(* PLC project flexManufacturing.project, CODESYS CODESYS V3.5 SP16 Patch 3 *)
(* stored: creationDateTime 2021-01-27T23:10:48.5476869, modificationDateTime 2021-01-27T23:10:24.2476033 *)

PROGRAM PLC_PRG
  VAR
    FM_CPS_PP_DETECTED : BOOL;  (* INPUTS *)
    FM_CPS_PP_MOVINGX : BOOL;
    FM_CPS_PP_MOVINGZ : BOOL;
    FM_CPS_PP_ROTATING : BOOL;
    FM_CPS_TRANSFER_END : BOOL;
    FM_INPUT_1_SENSOR : BOOL;
    FM_INPUT_2_SENSOR : BOOL;
    FM_PALLET_1_CONV_1_END : BOOL;
    FM_PALLET_1_CONV_2_END : BOOL;
    FM_PALLET_2_CONV_1_END : BOOL;
    FM_PALLET_2_CONV_6_END : BOOL;
    FM_PALLET_3_CONV_1_END : BOOL;
    FM_PALLET_3_CONV_2_END : BOOL;
    FM_PALLET_4_CONV_1_END : BOOL;
    FM_PALLET_4_CONV_4_END : BOOL;
    FM_PALLET_5_CONV_1_END : BOOL;
    FM_PALLET_5_CONV_3_END : BOOL;
    FM_PALLET_2_CONV_2_3_SENSOR : BOOL;
    FM_PALLET_2_CONV_4_5_SENSOR : BOOL;
    FM_PALLET_4_CONV_2_3_SENSOR : BOOL;
    FM_PALLET_5_CONV_2_3_SENSOR : BOOL;
    FM_WS_1_M_BUSY : BOOL;
    FM_WS_2_M_BUSY : BOOL;
    FM_WS_1_PP_1_MOVINGX : BOOL;
    FM_WS_1_PP_1_MOVINGZ : BOOL;
    FM_WS_1_PP_2_MOVINGX : BOOL;
    FM_WS_1_PP_2_MOVINGZ : BOOL;
    FM_WS_2_PP_1_MOVINGX : BOOL;
    FM_WS_2_PP_1_MOVINGZ : BOOL;
    FM_WS_2_PP_2_MOVINGX : BOOL;
    FM_WS_2_PP_2_MOVINGZ : BOOL;
    FM_WS_3_PP_1_MOVINGX : BOOL;
    FM_WS_3_PP_1_MOVINGZ : BOOL;
    FM_WS_3_PP_2_MOVINGX : BOOL;
    FM_WS_3_PP_2_MOVINGZ : BOOL;
    FM_WS_3_PP_3_MOVINGX : BOOL;
    FM_WS_3_PP_3_MOVINGZ : BOOL;
    FM_WS_3_PP_4_MOVINGX : BOOL;
    FM_WS_3_PP_4_MOVINGZ : BOOL;
    FM_WS_1_PP_1_DETECTED : BOOL;
    FM_WS_1_PP_1_ROTATING : BOOL;
    FM_WS_1_PP_2_DETECTED : BOOL;
    FM_WS_1_PP_2_ROTATING : BOOL;
    FM_WS_2_PP_1_DETECTED : BOOL;
    FM_WS_2_PP_1_ROTATING : BOOL;
    FM_WS_2_PP_2_DETECTED : BOOL;
    FM_WS_2_PP_2_ROTATING : BOOL;
    FM_WS_3_PP_1_DETECTED : BOOL;
    FM_WS_3_PP_1_ROTATING : BOOL;
    FM_WS_3_PP_2_DETECTED : BOOL;
    FM_WS_3_PP_2_ROTATING : BOOL;
    FM_WS_3_PP_3_DETECTED : BOOL;
    FM_WS_3_PP_3_ROTATING : BOOL;
    FM_WS_3_PP_4_DETECTED : BOOL;
    FM_WS_3_PP_4_ROTATING : BOOL;
    FM_ZONE_1_SENSOR_1 : BOOL;
    FM_ZONE_1_SENSOR_2 : BOOL;
    FM_ZONE_2_SENSOR_1 : BOOL;
    FM_ZONE_2_SENSOR_2 : BOOL;
    FM_ZONE_3_SENSOR_1 : BOOL;
    FM_ZONE_3_SENSOR_2 : BOOL;
    FM_ZONE_4_SENSOR_1 : BOOL;
    FM_ZONE_4_SENSOR_2 : BOOL;
    FM_WS_3_CONV_PROD_END : BOOL;
    FM_CPS_CONV_F : BOOL;  (* OUTPUTS *)
    FM_CPS_INBOX_F : BOOL;
    FM_CPS_INBOX_WARNINGL : BOOL;
    FM_CPS_OUT_WARNINGl : BOOL;
    FM_CPS_PP_GRAB : BOOL;
    FM_CPS_PP_MOVX : BOOL;
    FM_CPS_PP_MOVZ : BOOL;
    FM_CPS_PP_ROTCW : BOOL;
    FM_CPS_PP_ROTCCW : BOOL;
    FM_CPS_TRANSFER_F : BOOL;
    FM_CPS_TRANSFER_R : BOOL;
    FM_INPUT_1 : BOOL;
    FM_INPUT_2 : BOOL;
    FM_INPUT_1_WARNINGL : BOOL;
    FM_INPUT_2_WARNINGL : BOOL;
    FM_PALLET_1_CONV_1_B : BOOL;
    FM_PALLET_1_CONV_1_F : BOOL;
    FM_PALLET_1_CONV_2_B : BOOL;
    FM_PALLET_1_CONV_2_F : BOOL;
    FM_PALLET_2_CONV_1_B : BOOL;
    FM_PALLET_2_CONV_1_F : BOOL;
    FM_PALLET_2_CONV_2_B : BOOL;
    FM_PALLET_2_CONV_2_F : BOOL;
    FM_PALLET_2_CONV_3_B : BOOL;
    FM_PALLET_2_CONV_3_F : BOOL;
    FM_PALLET_2_CONV_6_B : BOOL;
    FM_PALLET_2_CONV_6_F : BOOL;
    FM_PALLET_3_CONV_1_B : BOOL;
    FM_PALLET_3_CONV_1_F : BOOL;
    FM_PALLET_3_CONV_2_B : BOOL;
    FM_PALLET_3_CONV_2_F : BOOL;
    FM_PALLET_4_CONV_1_B : BOOL;
    FM_PALLET_4_CONV_1_F : BOOL;
    FM_PALLET_5_CONV_3_B : BOOL;
    FM_PALLET_5_CONV_3_F : BOOL;
    FM_PALLET_2_CONV_4_B_0 : BOOL;
    FM_PALLET_2_CONV_4_B_1 : BOOL;
    FM_PALLET_2_CONV_4_B_2 : BOOL;
    FM_PALLET_2_CONV_4_F_0 : BOOL;
    FM_PALLET_2_CONV_4_F_1 : BOOL;
    FM_PALLET_2_CONV_4_F_2 : BOOL;
    FM_PALLET_2_CONV_5_B_0 : BOOL;
    FM_PALLET_2_CONV_5_B_1 : BOOL;
    FM_PALLET_2_CONV_5_B_2 : BOOL;
    FM_PALLET_2_CONV_5_F_0 : BOOL;
    FM_PALLET_2_CONV_5_F_1 : BOOL;
    FM_PALLET_2_CONV_5_F_2 : BOOL;
    FM_PALLET_4_CONV_2_B_0 : BOOL;
    FM_PALLET_4_CONV_2_B_1 : BOOL;
    FM_PALLET_4_CONV_2_B_2 : BOOL;
    FM_PALLET_4_CONV_2_F_0 : BOOL;
    FM_PALLET_4_CONV_2_F_1 : BOOL;
    FM_PALLET_4_CONV_2_F_2 : BOOL;
    FM_PALLET_4_CONV_3_B_0 : BOOL;
    FM_PALLET_4_CONV_3_B_1 : BOOL;
    FM_PALLET_4_CONV_3_B_2 : BOOL;
    FM_PALLET_4_CONV_3_F_0 : BOOL;
    FM_PALLET_4_CONV_3_F_1 : BOOL;
    FM_PALLET_4_CONV_3_F_2 : BOOL;
    FM_PALLET_4_CONV_4_B_0 : BOOL;
    FM_PALLET_4_CONV_4_B_1 : BOOL;
    FM_PALLET_4_CONV_4_B_2 : BOOL;
    FM_PALLET_4_CONV_4_F_0 : BOOL;
    FM_PALLET_4_CONV_4_F_1 : BOOL;
    FM_PALLET_4_CONV_4_F_2 : BOOL;
    FM_PALLET_5_CONV_1_B_0 : BOOL;
    FM_PALLET_5_CONV_1_B_1 : BOOL;
    FM_PALLET_5_CONV_1_B_2 : BOOL;
    FM_PALLET_5_CONV_1_F_0 : BOOL;
    FM_PALLET_5_CONV_1_F_1 : BOOL;
    FM_PALLET_5_CONV_1_F_2 : BOOL;
    FM_PALLET_5_CONV_2_B_0 : BOOL;
    FM_PALLET_5_CONV_2_B_1 : BOOL;
    FM_PALLET_5_CONV_2_F_0 : BOOL;
    FM_PALLET_5_CONV_2_F_1 : BOOL;
    FM_WS_1_M_START : BOOL;
    FM_WS_2_M_START : BOOL;
    FM_WS_1_WARNINGL : BOOL;
    FM_WS_2_WARNINGL : BOOL;
    FM_WS_1_PP_1_GRAB : BOOL;
    FM_WS_1_PP_1_MOVX : BOOL;
    FM_WS_1_PP_1_MOVZ : BOOL;
    FM_WS_1_PP_2_GRAB : BOOL;
    FM_WS_1_PP_2_MOVX : BOOL;
    FM_WS_1_PP_2_MOVZ : BOOL;
    FM_WS_2_PP_1_GRAB : BOOL;
    FM_WS_2_PP_1_MOVX : BOOL;
    FM_WS_2_PP_1_MOVZ : BOOL;
    FM_WS_2_PP_2_GRAB : BOOL;
    FM_WS_2_PP_2_MOVX : BOOL;
    FM_WS_2_PP_2_MOVZ : BOOL;
    FM_WS_3_CONV_PROD : BOOL;
    FM_WS_3_PP_1_GRAB : BOOL;
    FM_WS_3_PP_1_MOVX : BOOL;
    FM_WS_3_PP_1_MOVZ : BOOL;
    FM_WS_3_PP_2_GRAB : BOOL;
    FM_WS_3_PP_2_MOVX : BOOL;
    FM_WS_3_PP_2_MOVZ : BOOL;
    FM_WS_3_PP_3_GRAB : BOOL;
    FM_WS_3_PP_3_MOVX : BOOL;
    FM_WS_3_PP_3_MOVZ : BOOL;
    FM_WS_3_PP_4_GRAB : BOOL;
    FM_WS_3_PP_4_MOVX : BOOL;
    FM_WS_3_PP_4_MOVZ : BOOL;
    FM_WS_1_PP_1_ROTCW : BOOL;
    FM_WS_1_PP_2_ROTCW : BOOL;
    FM_WS_2_PP_1_ROTCW : BOOL;
    FM_WS_2_PP_2_ROTCW : BOOL;
    FM_WS_3_CONV_LID_0 : BOOL;
    FM_WS_3_CONV_LID_1 : BOOL;
    FM_WS_3_CONV_LID_2 : BOOL;
    FM_WS_3_CONV_LID_END : BOOL;
    FM_WS_3_PP_1_ROTCW : BOOL;
    FM_WS_3_PP_2_ROTCW : BOOL;
    FM_WS_3_PP_3_ROTCW : BOOL;
    FM_WS_3_PP_4_ROTCW : BOOL;
    FM_WS_1_PP_1_ROTCCW : BOOL;
    FM_WS_1_PP_2_ROTCCW : BOOL;
    FM_WS_2_PP_1_ROTCCW : BOOL;
    FM_WS_2_PP_2_ROTCCW : BOOL;
    FM_WS_3_CONV_BASE_0 : BOOL;
    FM_WS_3_CONV_BASE_1 : BOOL;
    FM_WS_3_CONV_BASE_2 : BOOL;
    FM_WS_3_CONV_BASE_3 : BOOL;
    FM_WS_3_CONV_BASE_END : BOOL;
    FM_WS_3_PP_1_ROTCCW : BOOL;
    FM_WS_3_PP_2_ROTCCW : BOOL;
    FM_WS_3_PP_3_ROTCCW : BOOL;
    FM_WS_3_PP_4_ROTCCW : BOOL;
    WS_1_PP_1_FALLEDGE : F_TRIG;
    WS_1_PP_1_STEP : INT := 0;
    WS_1_PP_1_TON : TON;
    WS_1_PP_2_FALLEDGE : F_TRIG;
    WS_1_PP_2_STEP : INT := 0;
    WS_1_PP_2_TON : TON;
    WS_2_PP_1_FALLEDGE : F_TRIG;
    WS_2_PP_1_STEP : INT := 0;
    WS_2_PP_1_TON : TON;
    WS_2_PP_2_FALLEDGE : F_TRIG;
    WS_2_PP_2_STEP : INT := 0;
    WS_2_PP_2_TON : TON;
    WS_3_PP_1_FALLEDGE : F_TRIG;
    WS_3_PP_1_STEP : INT := 0;
    WS_3_PP_1_TON : TON;
    WS_3_PP_2_FALLEDGE : F_TRIG;
    WS_3_PP_2_STEP : INT := 0;
    WS_3_PP_2_TON : TON;
    WS_3_PP_3_FALLEDGE : F_TRIG;
    WS_3_PP_3_STEP : INT := 0;
    WS_3_PP_3_TON : TON;
    WS_3_PP_4_FALLEDGE : F_TRIG;
    WS_3_PP_4_STEP : INT := 0;
    WS_3_PP_4_TON : TON;
    WS_3_RESET_FALLEDGE : F_TRIG;
    WS_3_RESET_STEP : INT := 0;
    WS_3_RESET_TON : TON;
    CPS_PP_FALLEDGE : F_TRIG;
    CPS_PP_STEP : INT := 0;
    CPS_PP_TON : TON;
    CPS_RESET_FALLEDGE : F_TRIG;
    CPS_RESET_STEP : INT := 0;
    CPS_RESET_TON : TON;
    P_1_CONV_1_END_F : F_TRIG;
    P_1_CONV_2_END_F : F_TRIG;
    P_2_CONV_1_END_F : F_TRIG;
    P_2_CONV_6_END_F : F_TRIG;
    P_3_CONV_1_END_F : F_TRIG;
    TR_T3 : BOOL;
    TR_T2 : BOOL;
    TR_T7 : BOOL;
    TR_T10 : BOOL;
    TR_T11 : BOOL;
    TR_T6 : BOOL;
    TR_T15 : BOOL;
    TR_T14 : BOOL;
    TR_T19 : BOOL;
    TR_T18 : BOOL;
  END_VAR

(* transition INPUT_1_TR_FALL *)
                        P_1_CONV_1_END_F(CLK:=FM_PALLET_1_CONV_1_END);
INPUT_1_TR_FALL:=P_1_CONV_1_END_F.Q;
                      
(* transition P_1_C_2_END_TR_F *)
                        P_1_CONV_2_END_F(CLK:=FM_PALLET_1_CONV_2_END);
P_1_C_2_END_TR_F:=P_1_CONV_2_END_F.Q;
                      
(* transition P_2_C_6_END_TR_F *)
                        P_2_CONV_6_END_F(CLK:=FM_PALLET_2_CONV_6_END);
P_2_C_6_END_TR_F:=P_2_CONV_6_END_F.Q;
                      
(* transition INPUT_2_TR_FALL *)
                        P_2_CONV_1_END_F(CLK:=FM_PALLET_2_CONV_1_END);
INPUT_2_TR_FALL:=P_2_CONV_1_END_F.Q;
                      
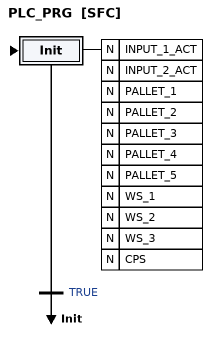
INITIAL_STEP Init:
  INPUT_1_ACT(N);
  INPUT_2_ACT(N);
  PALLET_1(N);
  PALLET_2(N);
  PALLET_3(N);
  PALLET_4(N);
  PALLET_5(N);
  WS_1(N);
  WS_2(N);
  WS_3(N);
  CPS(N);
END_STEP
TRANSITION FROM Init TO Init
  := TRUE;
END_TRANSITION

ACTION WS_1_ACT_PP_1:
                        
CASE WS_1_PP_1_STEP OF
	
	0:	FM_WS_1_PP_1_MOVX:=TRUE;
		WS_1_PP_1_STEP:=1;
		
	1:	FM_WS_1_PP_1_ROTCW:=TRUE;
		WS_1_PP_1_STEP:=2;
	
	2:	WS_1_PP_1_FALLEDGE(CLK:=FM_WS_1_PP_1_ROTATING);
		WHILE WS_1_PP_1_FALLEDGE.Q DO
			FM_WS_1_PP_1_MOVZ:=TRUE;
			WS_1_PP_1_STEP:=3;
			WS_1_PP_1_FALLEDGE(CLK:=FALSE);
		END_WHILE
		
	3:	FM_WS_1_PP_1_GRAB:=TRUE;
		WS_1_PP_1_STEP:=4;
		
	4:	WS_1_PP_1_FALLEDGE(CLK:=FM_WS_1_PP_1_MOVINGZ);
		WHILE WS_1_PP_1_FALLEDGE.Q DO
			FM_WS_1_PP_1_MOVZ:=FALSE;
			WS_1_PP_1_STEP:=5;
			WS_1_PP_1_FALLEDGE(CLK:=FALSE);
		END_WHILE
		
	5:	WS_1_PP_1_FALLEDGE(CLK:=FM_WS_1_PP_1_MOVINGZ);
		WHILE WS_1_PP_1_FALLEDGE.Q DO
			FM_WS_1_PP_1_ROTCCW:=TRUE;
			WS_1_PP_1_STEP:=6;
			WS_1_PP_1_FALLEDGE(CLK:=FALSE);
		END_WHILE
		
	6:	WS_1_PP_1_FALLEDGE(CLK:=FM_WS_1_PP_1_ROTATING);
		WHILE WS_1_PP_1_FALLEDGE.Q DO
			WS_1_PP_1_STEP:=7;
			WS_1_PP_1_FALLEDGE(CLK:=FALSE);
		END_WHILE
		
	7:	WS_1_PP_1_TON(IN:=TRUE,PT:=T#1S);
		WHILE WS_1_PP_1_TON.Q DO
			FM_WS_1_PP_1_GRAB:=FALSE;
			WS_1_PP_1_STEP:=8;
			WS_1_PP_1_TON(IN:=FALSE);
		END_WHILE
		
	8:	WS_1_PP_1_TON(IN:=TRUE,PT:=T#1S);
		WHILE WS_1_PP_1_TON.Q DO
			WS_1_PP_1_STEP:=9;
			WS_1_PP_1_TON(IN:=FALSE);
		END_WHILE
		
	9:	WS_1_PP_1_STEP:=0;
	
END_CASE

                      
END_ACTION

ACTION WS_1:
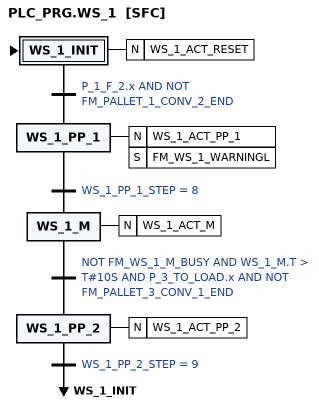
INITIAL_STEP WS_1_INIT:
  WS_1_ACT_RESET(N);
END_STEP
TRANSITION FROM WS_1_INIT TO WS_1_PP_1
  := P_1_F_2.x AND NOT FM_PALLET_1_CONV_2_END;
END_TRANSITION
STEP WS_1_PP_1:
  WS_1_ACT_PP_1(N);
  FM_WS_1_WARNINGL(S);
END_STEP
TRANSITION FROM WS_1_PP_1 TO WS_1_M
  := WS_1_PP_1_STEP = 8;
END_TRANSITION
STEP WS_1_M:
  WS_1_ACT_M(N);
END_STEP
TRANSITION FROM WS_1_M TO WS_1_PP_2
  := NOT FM_WS_1_M_BUSY AND WS_1_M.T > T#10S AND P_3_TO_LOAD.x AND NOT FM_PALLET_3_CONV_1_END;
END_TRANSITION
STEP WS_1_PP_2:
  WS_1_ACT_PP_2(N);
END_STEP
TRANSITION FROM WS_1_PP_2 TO WS_1_INIT
  := WS_1_PP_2_STEP = 9;
END_TRANSITION
END_ACTION

ACTION WS_1_ACT_PP_2:
                        
CASE WS_1_PP_2_STEP OF
	
	0:	FM_WS_1_PP_2_MOVX:=TRUE;
		WS_1_PP_2_STEP:=1;
		
	1:	WS_1_PP_2_FALLEDGE(CLK:=FM_WS_1_PP_2_MOVINGX);
		WHILE WS_1_PP_2_FALLEDGE.Q DO
			FM_WS_1_PP_2_MOVZ:=TRUE;
			WS_1_PP_2_STEP:=2;
			WS_1_PP_2_FALLEDGE(CLK:=FALSE);
		END_WHILE
		
	2:	FM_WS_1_PP_2_GRAB:=TRUE;
		WS_1_PP_2_STEP:=3;
		
	3:	WS_1_PP_2_FALLEDGE(CLK:=FM_WS_1_PP_2_MOVINGZ);
		WHILE WS_1_PP_2_FALLEDGE.Q DO
			FM_WS_1_PP_2_MOVZ:=FALSE;
			WS_1_PP_2_STEP:=4;
			WS_1_PP_2_FALLEDGE(CLK:=FALSE);
		END_WHILE
		
	4:	WS_1_PP_2_FALLEDGE(CLK:=FM_WS_1_PP_2_MOVINGZ);
		WHILE WS_1_PP_2_FALLEDGE.Q DO
			FM_WS_1_PP_2_ROTCCW:=TRUE;
			WS_1_PP_2_STEP:=5;
			WS_1_PP_2_FALLEDGE(CLK:=FALSE);
		END_WHILE
		
	5:	WS_1_PP_2_FALLEDGE(CLK:=FM_WS_1_PP_2_ROTATING);
		WHILE WS_1_PP_2_FALLEDGE.Q DO
			WS_1_PP_2_STEP:=6;
			FM_WS_1_PP_2_ROTCCW:=FALSE;
			WS_1_PP_2_FALLEDGE(CLK:=FALSE);
		END_WHILE
		
	6:	WS_1_PP_2_TON(IN:=TRUE,PT:=T#1S);
		WHILE WS_1_PP_2_TON.Q DO
			FM_WS_1_PP_2_GRAB:=FALSE;
			WS_1_PP_2_STEP:=7;
			WS_1_PP_2_TON(IN:=FALSE);
		END_WHILE
		
	7:	WS_1_PP_2_TON(IN:=TRUE,PT:=T#1S);
		WHILE WS_1_PP_2_TON.Q DO
			FM_WS_1_PP_2_ROTCW:=TRUE;
			WS_1_PP_2_STEP:=8;
			WS_1_PP_2_TON(IN:=FALSE);
		END_WHILE
		
	8:	WS_1_PP_2_FALLEDGE(CLK:=FM_WS_1_PP_2_ROTATING);
		WHILE WS_1_PP_2_FALLEDGE.Q DO
			WS_1_PP_2_STEP:=9;
			FM_WS_1_PP_2_ROTCW:=FALSE;
			WS_1_PP_2_FALLEDGE(CLK:=FALSE);
		END_WHILE
		
	9: WS_1_PP_2_STEP:=0;
END_CASE
                      
END_ACTION

ACTION WS_1_ACT_M:
                        FM_WS_1_M_START:=TRUE;
                      
END_ACTION

ACTION WS_1_ACT_RESET:
                        FM_WS_1_PP_1_MOVX:=FALSE;
FM_WS_1_PP_1_ROTCCW:=FALSE;
FM_WS_1_PP_1_ROTCW:=FALSE;
FM_WS_1_M_START:=FALSE;
FM_WS_1_WARNINGL:=FALSE;
FM_WS_1_PP_2_MOVX:=FALSE;
FM_WS_1_PP_2_ROTCCW:=FALSE;
FM_WS_1_PP_2_ROTCW:=FALSE;

                      
END_ACTION

ACTION WS_3:
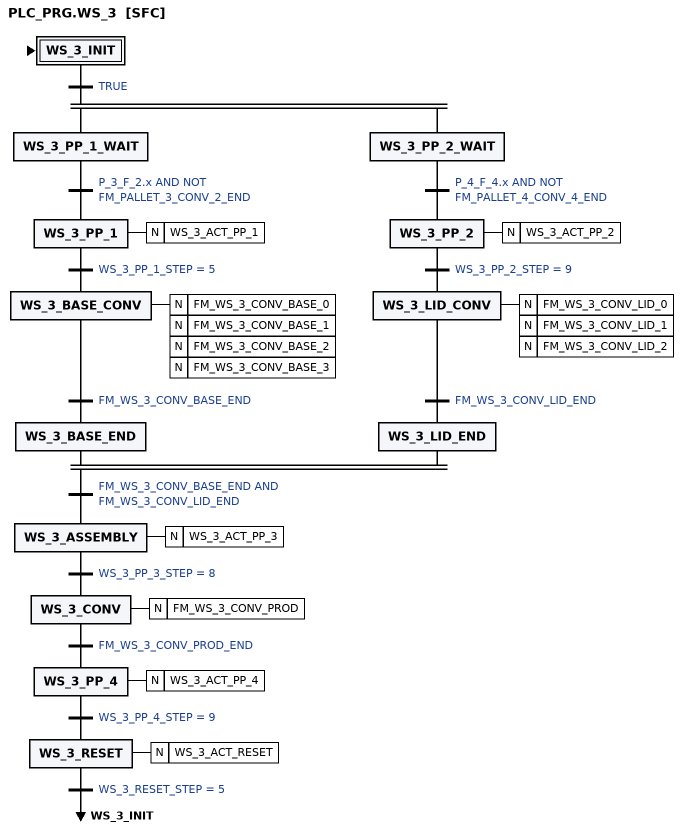
INITIAL_STEP WS_3_INIT:
END_STEP
TRANSITION FROM WS_3_INIT TO (WS_3_PP_1_WAIT, WS_3_PP_2_WAIT)
  := TRUE;
END_TRANSITION
STEP WS_3_PP_1_WAIT:
END_STEP
TRANSITION FROM WS_3_PP_1_WAIT TO WS_3_PP_1
  := P_3_F_2.x AND NOT FM_PALLET_3_CONV_2_END;
END_TRANSITION
STEP WS_3_PP_1:
  WS_3_ACT_PP_1(N);
END_STEP
TRANSITION FROM WS_3_PP_1 TO WS_3_BASE_CONV
  := WS_3_PP_1_STEP = 5;
END_TRANSITION
STEP WS_3_BASE_CONV:
  FM_WS_3_CONV_BASE_0(N);
  FM_WS_3_CONV_BASE_1(N);
  FM_WS_3_CONV_BASE_2(N);
  FM_WS_3_CONV_BASE_3(N);
END_STEP
TRANSITION FROM WS_3_BASE_CONV TO WS_3_BASE_END
  := FM_WS_3_CONV_BASE_END;
END_TRANSITION
STEP WS_3_BASE_END:
END_STEP
TRANSITION FROM (WS_3_BASE_END, WS_3_LID_END) TO WS_3_ASSEMBLY
  := FM_WS_3_CONV_BASE_END AND FM_WS_3_CONV_LID_END;
END_TRANSITION
STEP WS_3_PP_2_WAIT:
END_STEP
TRANSITION FROM WS_3_PP_2_WAIT TO WS_3_PP_2
  := P_4_F_4.x AND NOT FM_PALLET_4_CONV_4_END;
END_TRANSITION
STEP WS_3_PP_2:
  WS_3_ACT_PP_2(N);
END_STEP
TRANSITION FROM WS_3_PP_2 TO WS_3_LID_CONV
  := WS_3_PP_2_STEP = 9;
END_TRANSITION
STEP WS_3_LID_CONV:
  FM_WS_3_CONV_LID_0(N);
  FM_WS_3_CONV_LID_1(N);
  FM_WS_3_CONV_LID_2(N);
END_STEP
TRANSITION FROM WS_3_LID_CONV TO WS_3_LID_END
  := FM_WS_3_CONV_LID_END;
END_TRANSITION
STEP WS_3_LID_END:
END_STEP
STEP WS_3_ASSEMBLY:
  WS_3_ACT_PP_3(N);
END_STEP
TRANSITION FROM WS_3_ASSEMBLY TO WS_3_CONV
  := WS_3_PP_3_STEP = 8;
END_TRANSITION
STEP WS_3_CONV:
  FM_WS_3_CONV_PROD(N);
END_STEP
TRANSITION FROM WS_3_CONV TO WS_3_PP_4
  := FM_WS_3_CONV_PROD_END;
END_TRANSITION
STEP WS_3_PP_4:
  WS_3_ACT_PP_4(N);
END_STEP
TRANSITION FROM WS_3_PP_4 TO WS_3_RESET
  := WS_3_PP_4_STEP = 9;
END_TRANSITION
STEP WS_3_RESET:
  WS_3_ACT_RESET(N);
END_STEP
TRANSITION FROM WS_3_RESET TO WS_3_INIT
  := WS_3_RESET_STEP = 5;
END_TRANSITION
END_ACTION

ACTION WS_3_ACT_PP_1:
                        
CASE WS_3_PP_1_STEP OF
	
	0:	FM_WS_3_PP_1_MOVZ:=TRUE;
		FM_WS_3_PP_1_GRAB:=TRUE;
		WS_3_PP_1_STEP:=1;
		
	1:	WS_3_PP_1_FALLEDGE(CLK:=FM_WS_3_PP_1_MOVINGZ);
		WHILE WS_3_PP_1_FALLEDGE.Q DO
			FM_WS_3_PP_1_MOVZ:=FALSE;
			WS_3_PP_1_STEP:=2;
			WS_3_PP_1_FALLEDGE(CLK:=FALSE);
		END_WHILE
	
	2:	WS_3_PP_1_FALLEDGE(CLK:=FM_WS_3_PP_1_MOVINGZ);
		WHILE WS_3_PP_1_FALLEDGE.Q DO
			FM_WS_3_PP_1_MOVX:=TRUE;
			WS_3_PP_1_STEP:=3;
			WS_3_PP_1_FALLEDGE(CLK:=FALSE);
		END_WHILE
		
	3:	WS_3_PP_1_FALLEDGE(CLK:=FM_WS_3_PP_1_MOVINGX);
		WHILE WS_3_PP_1_FALLEDGE.Q DO
			WS_3_PP_1_STEP:=4;
			WS_3_PP_1_FALLEDGE(CLK:=FALSE);
		END_WHILE
		
	4:	WS_3_PP_1_TON(IN:=TRUE,PT:=T#200MS);
		WHILE WS_3_PP_1_TON.Q DO
			FM_WS_3_PP_1_GRAB:=FALSE;
			WS_3_PP_1_STEP:=5;
			WS_3_PP_1_TON(IN:=FALSE);
		END_WHILE
		
	5:	WS_3_PP_1_STEP:=0;
	
END_CASE
                      
END_ACTION

ACTION WS_3_ACT_PP_2:
                        
CASE WS_3_PP_2_STEP OF
	
	0:	FM_WS_3_PP_2_MOVX:=TRUE;
		WS_3_PP_2_STEP:=1;
		
	1:	WS_3_PP_2_FALLEDGE(CLK:=FM_WS_3_PP_2_MOVINGX);
		WHILE WS_3_PP_2_FALLEDGE.Q DO
			FM_WS_3_PP_2_MOVZ:=TRUE;
			FM_WS_3_PP_2_GRAB:=TRUE;
			WS_3_PP_2_STEP:=2;
			WS_3_PP_2_FALLEDGE(CLK:=FALSE);
		END_WHILE
	
	2:	WS_3_PP_2_FALLEDGE(CLK:=FM_WS_3_PP_2_MOVINGZ);
		WHILE WS_3_PP_2_FALLEDGE.Q DO
			FM_WS_3_PP_2_MOVZ:=FALSE;
			WS_3_PP_2_STEP:=3;
			WS_3_PP_2_FALLEDGE(CLK:=FALSE);
		END_WHILE
		
	3:	WS_3_PP_2_FALLEDGE(CLK:=FM_WS_3_PP_2_MOVINGZ);
		WHILE WS_3_PP_2_FALLEDGE.Q DO
			FM_WS_3_PP_2_ROTCCW:=TRUE;
			WS_3_PP_2_STEP:=4;
			WS_3_PP_2_FALLEDGE(CLK:=FALSE);
		END_WHILE
		
	4:	WS_3_PP_2_FALLEDGE(CLK:=FM_WS_3_PP_2_ROTATING);
		WHILE WS_3_PP_2_FALLEDGE.Q DO
			FM_WS_3_PP_2_ROTCCW:=FALSE;
			WS_3_PP_2_STEP:=5;
			WS_3_PP_2_FALLEDGE(CLK:=FALSE);
		END_WHILE
	
	5:	WS_3_PP_2_TON(IN:=TRUE,PT:=T#250MS);
		WHILE WS_3_PP_2_TON.Q DO
			WS_3_PP_2_STEP:=6;
			WS_3_PP_2_TON(IN:=FALSE);
		END_WHILE
		
	6:	FM_WS_3_PP_2_ROTCCW:=TRUE;
		WS_3_PP_2_STEP:=7;
	
	7:	WS_3_PP_2_FALLEDGE(CLK:=FM_WS_3_PP_2_ROTATING);
		WHILE WS_3_PP_2_FALLEDGE.Q DO
			FM_WS_3_PP_2_ROTCCW:=FALSE;
			WS_3_PP_2_STEP:=8;
			WS_3_PP_2_FALLEDGE(CLK:=FALSE);
		END_WHILE
		
	8:	WS_3_PP_2_TON(IN:=TRUE,PT:=T#200MS);
		WHILE WS_3_PP_2_TON.Q DO
			FM_WS_3_PP_2_GRAB:=FALSE;
			WS_3_PP_2_STEP:=9;
			WS_3_PP_2_TON(IN:=FALSE);
		END_WHILE
		
	9:	WS_3_PP_2_STEP:=0;
	
END_CASE
                      
END_ACTION

ACTION WS_3_ACT_PP_3:
                        
CASE WS_3_PP_3_STEP OF
	
	0:	FM_WS_3_PP_3_MOVZ:=TRUE;
		FM_WS_3_PP_3_GRAB:=TRUE;
		WS_3_PP_3_STEP:=1;
		
	1:	WS_3_PP_3_FALLEDGE(CLK:=FM_WS_3_PP_3_MOVINGZ);
		WHILE WS_3_PP_3_FALLEDGE.Q DO
			FM_WS_3_PP_3_MOVZ:=FALSE;
			WS_3_PP_3_STEP:=2;
			WS_3_PP_3_FALLEDGE(CLK:=FALSE);
		END_WHILE
	
	2:	WS_3_PP_3_FALLEDGE(CLK:=FM_WS_3_PP_3_MOVINGZ);
		WHILE WS_3_PP_3_FALLEDGE.Q DO
			FM_WS_3_PP_3_MOVX:=TRUE;
			WS_3_PP_3_STEP:=3;
			WS_3_PP_3_FALLEDGE(CLK:=FALSE);
		END_WHILE
		
	3:	WS_3_PP_3_FALLEDGE(CLK:=FM_WS_3_PP_3_MOVINGX);
		WHILE WS_3_PP_3_FALLEDGE.Q DO
			FM_WS_3_PP_3_MOVZ:=TRUE;
			WS_3_PP_3_STEP:=4;
			WS_3_PP_3_FALLEDGE(CLK:=FALSE);
		END_WHILE
		
	4:	WS_3_PP_3_FALLEDGE(CLK:=FM_WS_3_PP_3_MOVINGZ);
		WHILE WS_3_PP_3_FALLEDGE.Q DO
			FM_WS_3_PP_3_MOVZ:=FALSE;
			WS_3_PP_3_STEP:=5;
			WS_3_PP_3_FALLEDGE(CLK:=FALSE);
		END_WHILE
	
	5:	WS_3_PP_3_FALLEDGE(CLK:=FM_WS_3_PP_3_MOVINGZ);
		WHILE WS_3_PP_3_FALLEDGE.Q DO
			FM_WS_3_PP_3_ROTCCW:=TRUE;
			WS_3_PP_3_STEP:=6;
			WS_3_PP_3_FALLEDGE(CLK:=FALSE);
		END_WHILE;
	
	6:	WS_3_PP_3_FALLEDGE(CLK:=FM_WS_3_PP_3_ROTATING);
		WHILE WS_3_PP_3_FALLEDGE.Q DO
			FM_WS_3_PP_3_ROTCCW:=FALSE;
			WS_3_PP_3_STEP:=7;
			WS_3_PP_3_FALLEDGE(CLK:=FALSE);
		END_WHILE
		
	7:	WS_3_PP_3_TON(IN:=TRUE,PT:=T#200MS);
		WHILE WS_3_PP_3_TON.Q DO
			FM_WS_3_PP_3_GRAB:=FALSE;
			WS_3_PP_3_STEP:=8;
			WS_3_PP_3_TON(IN:=FALSE);
		END_WHILE
		
	8:	WS_3_PP_3_STEP:=0;
	
END_CASE
                      
END_ACTION

ACTION WS_3_ACT_PP_4:
                        
CASE WS_3_PP_4_STEP OF
	
	0:	FM_WS_3_PP_4_MOVX:=TRUE;
		WS_3_PP_4_STEP:=1;
		
	1:	WS_3_PP_4_FALLEDGE(CLK:=FM_WS_3_PP_4_MOVINGX);
		WHILE WS_3_PP_4_FALLEDGE.Q DO
			FM_WS_3_PP_4_MOVZ:=TRUE;
			FM_WS_3_PP_4_GRAB:=TRUE;
			WS_3_PP_4_STEP:=2;
			WS_3_PP_4_FALLEDGE(CLK:=FALSE);
		END_WHILE
	
	2:	WS_3_PP_4_FALLEDGE(CLK:=FM_WS_3_PP_4_MOVINGZ);
		WHILE WS_3_PP_4_FALLEDGE.Q DO
			FM_WS_3_PP_4_MOVZ:=FALSE;
			WS_3_PP_4_STEP:=3;
			WS_3_PP_4_FALLEDGE(CLK:=FALSE);
		END_WHILE
		
	3:	WS_3_PP_4_FALLEDGE(CLK:=FM_WS_3_PP_4_MOVINGZ);
		WHILE WS_3_PP_4_FALLEDGE.Q DO
			FM_WS_3_PP_4_ROTCCW:=TRUE;
			WS_3_PP_4_STEP:=4;
			WS_3_PP_4_FALLEDGE(CLK:=FALSE);
		END_WHILE
		
	4:	WS_3_PP_4_FALLEDGE(CLK:=FM_WS_3_PP_4_ROTATING);
		WHILE WS_3_PP_4_FALLEDGE.Q DO
			FM_WS_3_PP_4_ROTCCW:=FALSE;
			WS_3_PP_4_STEP:=5;
			WS_3_PP_4_FALLEDGE(CLK:=FALSE);
		END_WHILE
	
	5:	WS_3_PP_4_TON(IN:=TRUE,PT:=T#250MS);
		WHILE WS_3_PP_4_TON.Q DO
			FM_WS_3_PP_4_ROTCCW:=TRUE;
			WS_3_PP_4_STEP:=6;
			WS_3_PP_4_TON(IN:=FALSE);
		END_WHILE
	
	6:	WS_3_PP_4_FALLEDGE(CLK:=FM_WS_3_PP_4_ROTATING);
		WHILE WS_3_PP_4_FALLEDGE.Q DO
			FM_WS_3_PP_4_ROTCCW:=FALSE;
			FM_WS_3_PP_4_MOVZ:=TRUE;
			WS_3_PP_4_STEP:=7;
			WS_3_PP_4_FALLEDGE(CLK:=FALSE);
		END_WHILE
		
	7:	WS_3_PP_4_FALLEDGE(CLK:=FM_WS_3_PP_4_MOVINGZ);
		WHILE WS_3_PP_4_FALLEDGE.Q DO
			FM_WS_3_PP_4_MOVZ:=FALSE;
			FM_WS_3_PP_4_GRAB:=FALSE;
			WS_3_PP_4_STEP:=8;
			WS_3_PP_4_FALLEDGE(CLK:=FALSE);
		END_WHILE
	
	8:	WS_3_PP_4_FALLEDGE(CLK:=FM_WS_3_PP_4_MOVINGZ);
		WHILE WS_3_PP_4_FALLEDGE.Q DO
			WS_3_PP_4_STEP:=9;
			WS_3_PP_4_FALLEDGE(CLK:=FALSE);
		END_WHILE	
		
	9:	WS_3_PP_4_STEP:=0;
	
END_CASE
                      
END_ACTION

ACTION WS_3_ACT_RESET:
                        
CASE WS_3_RESET_STEP OF
	
	0:	FM_WS_3_PP_1_MOVX:=FALSE;
		FM_WS_3_PP_2_MOVX:=FALSE;
		FM_WS_3_PP_2_ROTCW:=TRUE;
		FM_WS_3_PP_3_MOVX:=FALSE;
		FM_WS_3_PP_3_ROTCW:=TRUE;
		FM_WS_3_PP_4_MOVX:=FALSE;
		FM_WS_3_PP_4_ROTCW:=TRUE;
		WS_3_RESET_STEP:=1;
		
	1:	WS_3_RESET_FALLEDGE(CLK:=FM_WS_3_PP_2_ROTATING);
		WHILE WS_3_RESET_FALLEDGE.Q DO
			FM_WS_3_PP_2_ROTCW:=FALSE;
			FM_WS_3_PP_3_ROTCW:=FALSE;
			FM_WS_3_PP_4_ROTCW:=FALSE;
			WS_3_RESET_STEP:=2;
			WS_3_RESET_FALLEDGE(CLK:=FALSE);
		END_WHILE
	
	2:	WS_3_RESET_TON(IN:=TRUE,PT:=T#300MS);
		WHILE WS_3_RESET_TON.Q DO
			WS_3_RESET_STEP:=3;
			WS_3_RESET_TON(IN:=FALSE);
		END_WHILE
		
	3:	FM_WS_3_PP_2_ROTCW:=TRUE;
		FM_WS_3_PP_4_ROTCW:=TRUE;
		WS_3_RESET_STEP:=4;
	
	4:	WS_3_RESET_FALLEDGE(CLK:=FM_WS_3_PP_2_ROTATING);
		WHILE WS_3_RESET_FALLEDGE.Q DO
			FM_WS_3_PP_2_ROTCW:=FALSE;
			FM_WS_3_PP_4_ROTCW:=FALSE;
			WS_3_RESET_STEP:=5;
			WS_3_RESET_FALLEDGE(CLK:=FALSE);
		END_WHILE
		
	5:	WS_3_RESET_STEP:=0;
	
END_CASE
                      
END_ACTION

ACTION CPS:
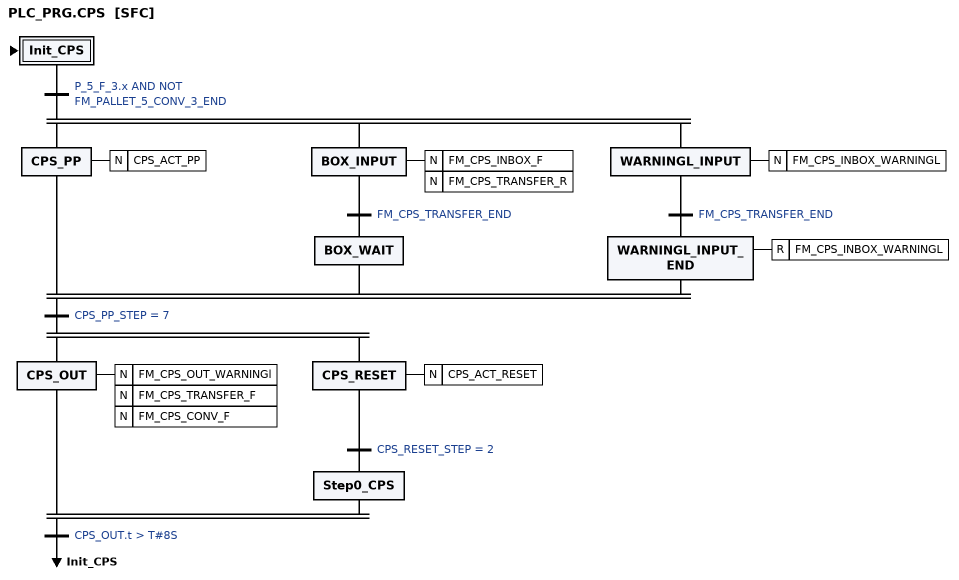
INITIAL_STEP Init_CPS:
END_STEP
TRANSITION FROM Init_CPS TO (CPS_PP, BOX_INPUT, WARNINGL_INPUT)
  := P_5_F_3.x AND NOT FM_PALLET_5_CONV_3_END;
END_TRANSITION
STEP CPS_PP:
  CPS_ACT_PP(N);
END_STEP
TRANSITION FROM (CPS_PP, BOX_WAIT, WARNINGL_INPUT_END) TO (CPS_OUT, CPS_RESET)
  := CPS_PP_STEP = 7;
END_TRANSITION
STEP BOX_INPUT:
  FM_CPS_INBOX_F(N);
  FM_CPS_TRANSFER_R(N);
END_STEP
TRANSITION FROM BOX_INPUT TO BOX_WAIT
  := FM_CPS_TRANSFER_END;
END_TRANSITION
STEP BOX_WAIT:
END_STEP
STEP WARNINGL_INPUT:
  FM_CPS_INBOX_WARNINGL(N);
END_STEP
TRANSITION FROM WARNINGL_INPUT TO WARNINGL_INPUT_END
  := FM_CPS_TRANSFER_END;
END_TRANSITION
STEP WARNINGL_INPUT_END:
  FM_CPS_INBOX_WARNINGL(R);
END_STEP
STEP CPS_OUT:
  FM_CPS_OUT_WARNINGl(N);
  FM_CPS_TRANSFER_F(N);
  FM_CPS_CONV_F(N);
END_STEP
TRANSITION FROM (CPS_OUT, Step0_CPS) TO Init_CPS
  := CPS_OUT.t > T#8S;
END_TRANSITION
STEP CPS_RESET:
  CPS_ACT_RESET(N);
END_STEP
TRANSITION FROM CPS_RESET TO Step0_CPS
  := CPS_RESET_STEP = 2;
END_TRANSITION
STEP Step0_CPS:
END_STEP
END_ACTION

ACTION CPS_ACT_PP:
                        
CASE CPS_PP_STEP OF
	
	0:	FM_CPS_PP_MOVX:=TRUE;
		CPS_PP_STEP:=1;
		
	1:	CPS_PP_FALLEDGE(CLK:=FM_CPS_PP_MOVINGX);
		WHILE CPS_PP_FALLEDGE.Q DO
			FM_CPS_PP_MOVZ:=TRUE;
			FM_CPS_PP_GRAB:=TRUE;
			CPS_PP_STEP:=2;
			CPS_PP_FALLEDGE(CLK:=FALSE);
		END_WHILE
	
	2:	CPS_PP_FALLEDGE(CLK:=FM_CPS_PP_MOVINGZ);
		WHILE CPS_PP_FALLEDGE.Q DO
			FM_CPS_PP_MOVZ:=FALSE;
			CPS_PP_STEP:=3;
			CPS_PP_FALLEDGE(CLK:=FALSE);
		END_WHILE
		
	3:	CPS_PP_FALLEDGE(CLK:=FM_CPS_PP_MOVINGZ);
		WHILE CPS_PP_FALLEDGE.Q DO
			FM_CPS_PP_ROTCW:=TRUE;
			CPS_PP_STEP:=4;
			CPS_PP_FALLEDGE(CLK:=FALSE);
		END_WHILE
		
	4:	CPS_PP_FALLEDGE(CLK:=FM_CPS_PP_ROTATING);
		WHILE CPS_PP_FALLEDGE.Q DO
			FM_CPS_PP_ROTCW:=FALSE;
			CPS_PP_STEP:=5;
			CPS_PP_FALLEDGE(CLK:=FALSE);
		END_WHILE
		
	5:	CPS_PP_TON(IN:=TRUE,PT:=T#300MS);
		WHILE CPS_PP_TON.Q DO
			FM_CPS_PP_GRAB:=FALSE;
			CPS_PP_STEP:=6;
			CPS_PP_TON(IN:=FALSE);
		END_WHILE
		
	6:	CPS_PP_TON(IN:=TRUE,PT:=T#500MS);
		WHILE CPS_PP_TON.Q DO
			CPS_PP_STEP:=7;
			CPS_PP_TON(IN:=FALSE);
		END_WHILE
		
	7:	CPS_PP_STEP:=0;
	
END_CASE
                      
END_ACTION

ACTION PALLET_3:
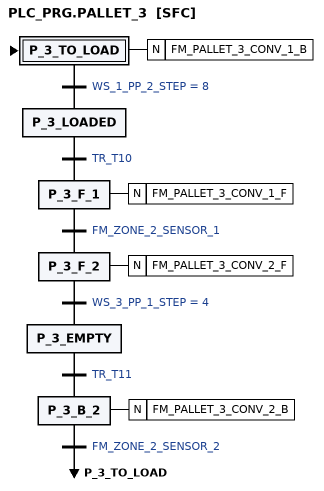
INITIAL_STEP P_3_TO_LOAD:
  FM_PALLET_3_CONV_1_B(N);
END_STEP
TRANSITION FROM P_3_TO_LOAD TO P_3_LOADED
  := WS_1_PP_2_STEP = 8;
END_TRANSITION
STEP P_3_LOADED:
END_STEP
TRANSITION FROM P_3_LOADED TO P_3_F_1
  := TR_T10;
END_TRANSITION
STEP P_3_F_1:
  FM_PALLET_3_CONV_1_F(N);
END_STEP
TRANSITION FROM P_3_F_1 TO P_3_F_2
  := FM_ZONE_2_SENSOR_1;
END_TRANSITION
STEP P_3_F_2:
  FM_PALLET_3_CONV_2_F(N);
END_STEP
TRANSITION FROM P_3_F_2 TO P_3_EMPTY
  := WS_3_PP_1_STEP = 4;
END_TRANSITION
STEP P_3_EMPTY:
END_STEP
TRANSITION FROM P_3_EMPTY TO P_3_B_2
  := TR_T11;
END_TRANSITION
STEP P_3_B_2:
  FM_PALLET_3_CONV_2_B(N);
END_STEP
TRANSITION FROM P_3_B_2 TO P_3_TO_LOAD
  := FM_ZONE_2_SENSOR_2;
END_TRANSITION
END_ACTION

ACTION WS_2_ACT_M:
                        FM_WS_2_M_START:=TRUE;
                      
END_ACTION

ACTION WS_2_ACT_PP_1:
                        
CASE WS_2_PP_1_STEP OF
	
	0:	FM_WS_2_PP_1_MOVX:=TRUE;
		WS_2_PP_1_STEP:=1;
		
	1:	FM_WS_2_PP_1_ROTCW:=TRUE;
		WS_2_PP_1_STEP:=2;
	
	2:	WS_2_PP_1_FALLEDGE(CLK:=FM_WS_2_PP_1_ROTATING);
		WHILE WS_2_PP_1_FALLEDGE.Q DO
			FM_WS_2_PP_1_MOVZ:=TRUE;
			WS_2_PP_1_STEP:=3;
			WS_2_PP_1_FALLEDGE(CLK:=FALSE);
		END_WHILE
		
	3:	FM_WS_2_PP_1_GRAB:=TRUE;
		WS_2_PP_1_STEP:=4;
		
	4:	WS_2_PP_1_FALLEDGE(CLK:=FM_WS_2_PP_1_MOVINGZ);
		WHILE WS_2_PP_1_FALLEDGE.Q DO
			FM_WS_2_PP_1_MOVZ:=FALSE;
			WS_2_PP_1_STEP:=5;
			WS_2_PP_1_FALLEDGE(CLK:=FALSE);
		END_WHILE
		
	5:	WS_2_PP_1_FALLEDGE(CLK:=FM_WS_2_PP_1_MOVINGZ);
		WHILE WS_2_PP_1_FALLEDGE.Q DO
			FM_WS_2_PP_1_ROTCCW:=TRUE;
			WS_2_PP_1_STEP:=6;
			WS_2_PP_1_FALLEDGE(CLK:=FALSE);
		END_WHILE
		
	6:	WS_2_PP_1_FALLEDGE(CLK:=FM_WS_2_PP_1_ROTATING);
		WHILE WS_2_PP_1_FALLEDGE.Q DO
			WS_2_PP_1_STEP:=7;
			WS_2_PP_1_FALLEDGE(CLK:=FALSE);
		END_WHILE
		
	7:	WS_2_PP_1_TON(IN:=TRUE,PT:=T#1S);
		WHILE WS_2_PP_1_TON.Q DO
			FM_WS_2_PP_1_GRAB:=FALSE;
			WS_2_PP_1_STEP:=8;
			WS_2_PP_1_TON(IN:=FALSE);
		END_WHILE
		
	8:	WS_2_PP_1_TON(IN:=TRUE,PT:=T#1S);
		WHILE WS_2_PP_1_TON.Q DO
			WS_2_PP_1_STEP:=9;
			WS_2_PP_1_TON(IN:=FALSE);
		END_WHILE
		
	9:	WS_2_PP_1_STEP:=0;
	
END_CASE

                      
END_ACTION

ACTION WS_2_ACT_PP_2:
                        
CASE WS_2_PP_2_STEP OF
	
	0:	FM_WS_2_PP_2_MOVX:=TRUE;
		WS_2_PP_2_STEP:=1;
		
	1:	WS_2_PP_2_FALLEDGE(CLK:=FM_WS_2_PP_2_MOVINGX);
		WHILE WS_2_PP_2_FALLEDGE.Q DO
			FM_WS_2_PP_2_MOVZ:=TRUE;
			WS_2_PP_2_STEP:=2;
			WS_2_PP_2_FALLEDGE(CLK:=FALSE);
		END_WHILE
		
	2:	FM_WS_2_PP_2_GRAB:=TRUE;
		WS_2_PP_2_STEP:=3;
		
	3:	WS_2_PP_2_FALLEDGE(CLK:=FM_WS_2_PP_2_MOVINGZ);
		WHILE WS_2_PP_2_FALLEDGE.Q DO
			FM_WS_2_PP_2_MOVZ:=FALSE;
			WS_2_PP_2_STEP:=4;
			WS_2_PP_2_FALLEDGE(CLK:=FALSE);
		END_WHILE
		
	4:	WS_2_PP_2_FALLEDGE(CLK:=FM_WS_2_PP_2_MOVINGZ);
		WHILE WS_2_PP_2_FALLEDGE.Q DO
			FM_WS_2_PP_2_ROTCCW:=TRUE;
			WS_2_PP_2_STEP:=5;
			WS_2_PP_2_FALLEDGE(CLK:=FALSE);
		END_WHILE
		
	5:	WS_2_PP_2_FALLEDGE(CLK:=FM_WS_2_PP_2_ROTATING);
		WHILE WS_2_PP_2_FALLEDGE.Q DO
			WS_2_PP_2_STEP:=6;
			FM_WS_2_PP_2_ROTCCW:=FALSE;
			WS_2_PP_2_FALLEDGE(CLK:=FALSE);
		END_WHILE
		
	6:	WS_2_PP_2_TON(IN:=TRUE,PT:=T#1S);
		WHILE WS_2_PP_2_TON.Q DO
			FM_WS_2_PP_2_GRAB:=FALSE;
			WS_2_PP_2_STEP:=7;
			WS_2_PP_2_TON(IN:=FALSE);
		END_WHILE
		
	7:	WS_2_PP_2_TON(IN:=TRUE,PT:=T#1S);
		WHILE WS_2_PP_2_TON.Q DO
			FM_WS_2_PP_2_ROTCW:=TRUE;
			WS_2_PP_2_STEP:=8;
			WS_2_PP_2_TON(IN:=FALSE);
		END_WHILE
		
	8:	WS_2_PP_2_FALLEDGE(CLK:=FM_WS_2_PP_2_ROTATING);
		WHILE WS_2_PP_2_FALLEDGE.Q DO
			WS_2_PP_2_STEP:=9;
			FM_WS_2_PP_2_ROTCW:=FALSE;
			WS_2_PP_2_FALLEDGE(CLK:=FALSE);
		END_WHILE
		
	9: WS_2_PP_2_STEP:=0;
END_CASE
                      
END_ACTION

ACTION WS_2_ACT_RESET:
                        FM_WS_2_PP_1_MOVX:=FALSE;
FM_WS_2_PP_1_ROTCCW:=FALSE;
FM_WS_2_PP_1_ROTCW:=FALSE;
FM_WS_2_M_START:=FALSE;
FM_WS_2_WARNINGL:=FALSE;
FM_WS_2_PP_2_MOVX:=FALSE;
FM_WS_2_PP_2_ROTCCW:=FALSE;
FM_WS_2_PP_2_ROTCW:=FALSE;

                      
END_ACTION

ACTION CPS_ACT_RESET:
                        CASE CPS_RESET_STEP OF
	
	0:	FM_CPS_PP_MOVX:=FALSE;
		FM_CPS_PP_ROTCCW:=TRUE;
		CPS_RESET_STEP:=1;
		
	1:	CPS_RESET_FALLEDGE(CLK:=FM_CPS_PP_ROTATING);
		WHILE CPS_RESET_FALLEDGE.Q DO
			FM_CPS_PP_ROTCCW:=FALSE;
			CPS_RESET_STEP:=2;
			CPS_RESET_FALLEDGE(CLK:=FALSE);
		END_WHILE
	
	2:	CPS_RESET_STEP:=0;
	
END_CASE
                      
END_ACTION

ACTION WS_2:
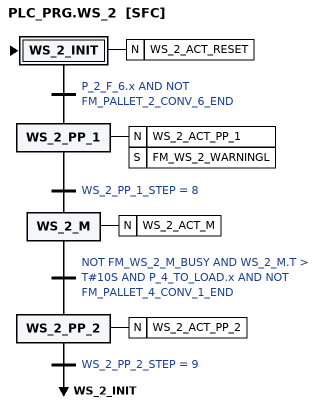
INITIAL_STEP WS_2_INIT:
  WS_2_ACT_RESET(N);
END_STEP
TRANSITION FROM WS_2_INIT TO WS_2_PP_1
  := P_2_F_6.x AND NOT FM_PALLET_2_CONV_6_END;
END_TRANSITION
STEP WS_2_PP_1:
  WS_2_ACT_PP_1(N);
  FM_WS_2_WARNINGL(S);
END_STEP
TRANSITION FROM WS_2_PP_1 TO WS_2_M
  := WS_2_PP_1_STEP = 8;
END_TRANSITION
STEP WS_2_M:
  WS_2_ACT_M(N);
END_STEP
TRANSITION FROM WS_2_M TO WS_2_PP_2
  := NOT FM_WS_2_M_BUSY AND WS_2_M.T > T#10S AND P_4_TO_LOAD.x AND NOT FM_PALLET_4_CONV_1_END;
END_TRANSITION
STEP WS_2_PP_2:
  WS_2_ACT_PP_2(N);
END_STEP
TRANSITION FROM WS_2_PP_2 TO WS_2_INIT
  := WS_2_PP_2_STEP = 9;
END_TRANSITION
END_ACTION

ACTION INPUT_1_ACT:
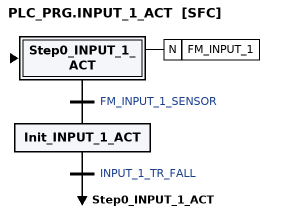
INITIAL_STEP Step0_INPUT_1_ACT:
  FM_INPUT_1(N);
END_STEP
TRANSITION FROM Step0_INPUT_1_ACT TO Init_INPUT_1_ACT
  := FM_INPUT_1_SENSOR;
END_TRANSITION
STEP Init_INPUT_1_ACT:
END_STEP
TRANSITION FROM Init_INPUT_1_ACT TO Step0_INPUT_1_ACT
  := INPUT_1_TR_FALL;
END_TRANSITION
END_ACTION

ACTION PALLET_1:
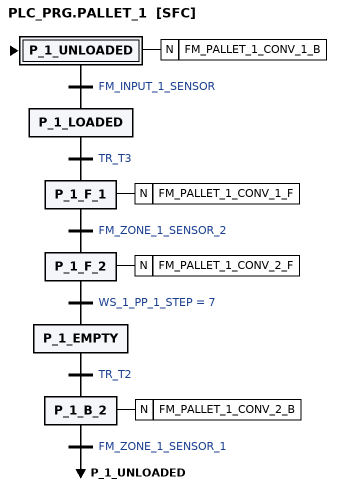
INITIAL_STEP P_1_UNLOADED:
  FM_PALLET_1_CONV_1_B(N);
END_STEP
TRANSITION FROM P_1_UNLOADED TO P_1_LOADED
  := FM_INPUT_1_SENSOR;
END_TRANSITION
STEP P_1_LOADED:
END_STEP
TRANSITION FROM P_1_LOADED TO P_1_F_1
  := TR_T3;
END_TRANSITION
STEP P_1_F_1:
  FM_PALLET_1_CONV_1_F(N);
END_STEP
TRANSITION FROM P_1_F_1 TO P_1_F_2
  := FM_ZONE_1_SENSOR_2;
END_TRANSITION
STEP P_1_F_2:
  FM_PALLET_1_CONV_2_F(N);
END_STEP
TRANSITION FROM P_1_F_2 TO P_1_EMPTY
  := WS_1_PP_1_STEP = 7;
END_TRANSITION
STEP P_1_EMPTY:
END_STEP
TRANSITION FROM P_1_EMPTY TO P_1_B_2
  := TR_T2;
END_TRANSITION
STEP P_1_B_2:
  FM_PALLET_1_CONV_2_B(N);
END_STEP
TRANSITION FROM P_1_B_2 TO P_1_UNLOADED
  := FM_ZONE_1_SENSOR_1;
END_TRANSITION
END_ACTION

ACTION PALLET_2:
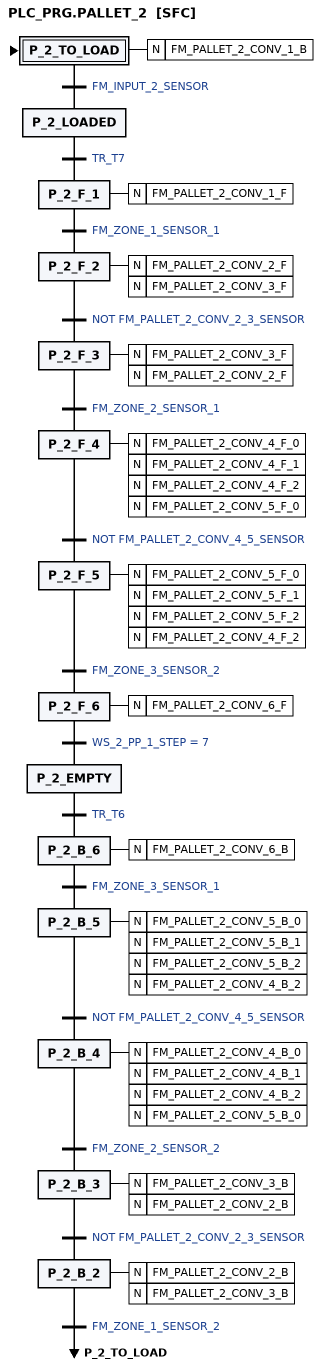
INITIAL_STEP P_2_TO_LOAD:
  FM_PALLET_2_CONV_1_B(N);
END_STEP
TRANSITION FROM P_2_TO_LOAD TO P_2_LOADED
  := FM_INPUT_2_SENSOR;
END_TRANSITION
STEP P_2_LOADED:
END_STEP
TRANSITION FROM P_2_LOADED TO P_2_F_1
  := TR_T7;
END_TRANSITION
STEP P_2_F_1:
  FM_PALLET_2_CONV_1_F(N);
END_STEP
TRANSITION FROM P_2_F_1 TO P_2_F_2
  := FM_ZONE_1_SENSOR_1;
END_TRANSITION
STEP P_2_F_2:
  FM_PALLET_2_CONV_2_F(N);
  FM_PALLET_2_CONV_3_F(N);
END_STEP
TRANSITION FROM P_2_F_2 TO P_2_F_3
  := NOT FM_PALLET_2_CONV_2_3_SENSOR;
END_TRANSITION
STEP P_2_F_3:
  FM_PALLET_2_CONV_3_F(N);
  FM_PALLET_2_CONV_2_F(N);
END_STEP
TRANSITION FROM P_2_F_3 TO P_2_F_4
  := FM_ZONE_2_SENSOR_1;
END_TRANSITION
STEP P_2_F_4:
  FM_PALLET_2_CONV_4_F_0(N);
  FM_PALLET_2_CONV_4_F_1(N);
  FM_PALLET_2_CONV_4_F_2(N);
  FM_PALLET_2_CONV_5_F_0(N);
END_STEP
TRANSITION FROM P_2_F_4 TO P_2_F_5
  := NOT FM_PALLET_2_CONV_4_5_SENSOR;
END_TRANSITION
STEP P_2_F_5:
  FM_PALLET_2_CONV_5_F_0(N);
  FM_PALLET_2_CONV_5_F_1(N);
  FM_PALLET_2_CONV_5_F_2(N);
  FM_PALLET_2_CONV_4_F_2(N);
END_STEP
TRANSITION FROM P_2_F_5 TO P_2_F_6
  := FM_ZONE_3_SENSOR_2;
END_TRANSITION
STEP P_2_F_6:
  FM_PALLET_2_CONV_6_F(N);
END_STEP
TRANSITION FROM P_2_F_6 TO P_2_EMPTY
  := WS_2_PP_1_STEP = 7;
END_TRANSITION
STEP P_2_EMPTY:
END_STEP
TRANSITION FROM P_2_EMPTY TO P_2_B_6
  := TR_T6;
END_TRANSITION
STEP P_2_B_6:
  FM_PALLET_2_CONV_6_B(N);
END_STEP
TRANSITION FROM P_2_B_6 TO P_2_B_5
  := FM_ZONE_3_SENSOR_1;
END_TRANSITION
STEP P_2_B_5:
  FM_PALLET_2_CONV_5_B_0(N);
  FM_PALLET_2_CONV_5_B_1(N);
  FM_PALLET_2_CONV_5_B_2(N);
  FM_PALLET_2_CONV_4_B_2(N);
END_STEP
TRANSITION FROM P_2_B_5 TO P_2_B_4
  := NOT FM_PALLET_2_CONV_4_5_SENSOR;
END_TRANSITION
STEP P_2_B_4:
  FM_PALLET_2_CONV_4_B_0(N);
  FM_PALLET_2_CONV_4_B_1(N);
  FM_PALLET_2_CONV_4_B_2(N);
  FM_PALLET_2_CONV_5_B_0(N);
END_STEP
TRANSITION FROM P_2_B_4 TO P_2_B_3
  := FM_ZONE_2_SENSOR_2;
END_TRANSITION
STEP P_2_B_3:
  FM_PALLET_2_CONV_3_B(N);
  FM_PALLET_2_CONV_2_B(N);
END_STEP
TRANSITION FROM P_2_B_3 TO P_2_B_2
  := NOT FM_PALLET_2_CONV_2_3_SENSOR;
END_TRANSITION
STEP P_2_B_2:
  FM_PALLET_2_CONV_2_B(N);
  FM_PALLET_2_CONV_3_B(N);
END_STEP
TRANSITION FROM P_2_B_2 TO P_2_TO_LOAD
  := FM_ZONE_1_SENSOR_2;
END_TRANSITION
END_ACTION

ACTION INPUT_2_ACT:
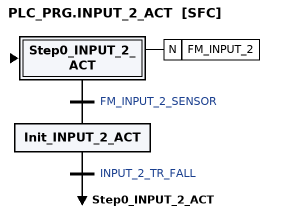
INITIAL_STEP Step0_INPUT_2_ACT:
  FM_INPUT_2(N);
END_STEP
TRANSITION FROM Step0_INPUT_2_ACT TO Init_INPUT_2_ACT
  := FM_INPUT_2_SENSOR;
END_TRANSITION
STEP Init_INPUT_2_ACT:
END_STEP
TRANSITION FROM Init_INPUT_2_ACT TO Step0_INPUT_2_ACT
  := INPUT_2_TR_FALL;
END_TRANSITION
END_ACTION

ACTION PALLET_4:
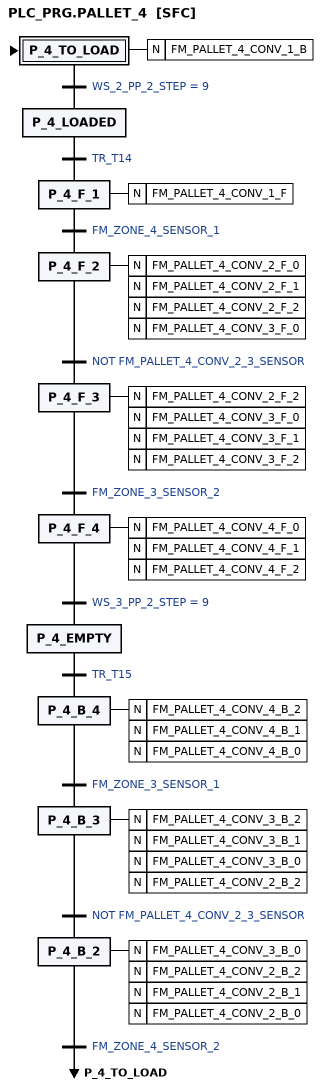
INITIAL_STEP P_4_TO_LOAD:
  FM_PALLET_4_CONV_1_B(N);
END_STEP
TRANSITION FROM P_4_TO_LOAD TO P_4_LOADED
  := WS_2_PP_2_STEP = 9;
END_TRANSITION
STEP P_4_LOADED:
END_STEP
TRANSITION FROM P_4_LOADED TO P_4_F_1
  := TR_T14;
END_TRANSITION
STEP P_4_F_1:
  FM_PALLET_4_CONV_1_F(N);
END_STEP
TRANSITION FROM P_4_F_1 TO P_4_F_2
  := FM_ZONE_4_SENSOR_1;
END_TRANSITION
STEP P_4_F_2:
  FM_PALLET_4_CONV_2_F_0(N);
  FM_PALLET_4_CONV_2_F_1(N);
  FM_PALLET_4_CONV_2_F_2(N);
  FM_PALLET_4_CONV_3_F_0(N);
END_STEP
TRANSITION FROM P_4_F_2 TO P_4_F_3
  := NOT FM_PALLET_4_CONV_2_3_SENSOR;
END_TRANSITION
STEP P_4_F_3:
  FM_PALLET_4_CONV_2_F_2(N);
  FM_PALLET_4_CONV_3_F_0(N);
  FM_PALLET_4_CONV_3_F_1(N);
  FM_PALLET_4_CONV_3_F_2(N);
END_STEP
TRANSITION FROM P_4_F_3 TO P_4_F_4
  := FM_ZONE_3_SENSOR_2;
END_TRANSITION
STEP P_4_F_4:
  FM_PALLET_4_CONV_4_F_0(N);
  FM_PALLET_4_CONV_4_F_1(N);
  FM_PALLET_4_CONV_4_F_2(N);
END_STEP
TRANSITION FROM P_4_F_4 TO P_4_EMPTY
  := WS_3_PP_2_STEP = 9;
END_TRANSITION
STEP P_4_EMPTY:
END_STEP
TRANSITION FROM P_4_EMPTY TO P_4_B_4
  := TR_T15;
END_TRANSITION
STEP P_4_B_4:
  FM_PALLET_4_CONV_4_B_2(N);
  FM_PALLET_4_CONV_4_B_1(N);
  FM_PALLET_4_CONV_4_B_0(N);
END_STEP
TRANSITION FROM P_4_B_4 TO P_4_B_3
  := FM_ZONE_3_SENSOR_1;
END_TRANSITION
STEP P_4_B_3:
  FM_PALLET_4_CONV_3_B_2(N);
  FM_PALLET_4_CONV_3_B_1(N);
  FM_PALLET_4_CONV_3_B_0(N);
  FM_PALLET_4_CONV_2_B_2(N);
END_STEP
TRANSITION FROM P_4_B_3 TO P_4_B_2
  := NOT FM_PALLET_4_CONV_2_3_SENSOR;
END_TRANSITION
STEP P_4_B_2:
  FM_PALLET_4_CONV_3_B_0(N);
  FM_PALLET_4_CONV_2_B_2(N);
  FM_PALLET_4_CONV_2_B_1(N);
  FM_PALLET_4_CONV_2_B_0(N);
END_STEP
TRANSITION FROM P_4_B_2 TO P_4_TO_LOAD
  := FM_ZONE_4_SENSOR_2;
END_TRANSITION
END_ACTION

ACTION PALLET_5:
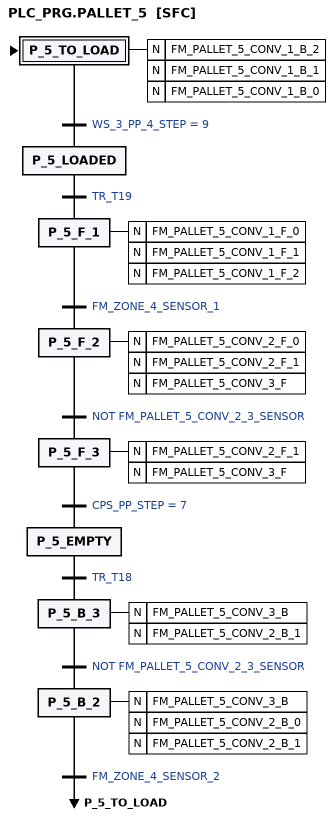
INITIAL_STEP P_5_TO_LOAD:
  FM_PALLET_5_CONV_1_B_2(N);
  FM_PALLET_5_CONV_1_B_1(N);
  FM_PALLET_5_CONV_1_B_0(N);
END_STEP
TRANSITION FROM P_5_TO_LOAD TO P_5_LOADED
  := WS_3_PP_4_STEP = 9;
END_TRANSITION
STEP P_5_LOADED:
END_STEP
TRANSITION FROM P_5_LOADED TO P_5_F_1
  := TR_T19;
END_TRANSITION
STEP P_5_F_1:
  FM_PALLET_5_CONV_1_F_0(N);
  FM_PALLET_5_CONV_1_F_1(N);
  FM_PALLET_5_CONV_1_F_2(N);
END_STEP
TRANSITION FROM P_5_F_1 TO P_5_F_2
  := FM_ZONE_4_SENSOR_1;
END_TRANSITION
STEP P_5_F_2:
  FM_PALLET_5_CONV_2_F_0(N);
  FM_PALLET_5_CONV_2_F_1(N);
  FM_PALLET_5_CONV_3_F(N);
END_STEP
TRANSITION FROM P_5_F_2 TO P_5_F_3
  := NOT FM_PALLET_5_CONV_2_3_SENSOR;
END_TRANSITION
STEP P_5_F_3:
  FM_PALLET_5_CONV_2_F_1(N);
  FM_PALLET_5_CONV_3_F(N);
END_STEP
TRANSITION FROM P_5_F_3 TO P_5_EMPTY
  := CPS_PP_STEP = 7;
END_TRANSITION
STEP P_5_EMPTY:
END_STEP
TRANSITION FROM P_5_EMPTY TO P_5_B_3
  := TR_T18;
END_TRANSITION
STEP P_5_B_3:
  FM_PALLET_5_CONV_3_B(N);
  FM_PALLET_5_CONV_2_B_1(N);
END_STEP
TRANSITION FROM P_5_B_3 TO P_5_B_2
  := NOT FM_PALLET_5_CONV_2_3_SENSOR;
END_TRANSITION
STEP P_5_B_2:
  FM_PALLET_5_CONV_3_B(N);
  FM_PALLET_5_CONV_2_B_0(N);
  FM_PALLET_5_CONV_2_B_1(N);
END_STEP
TRANSITION FROM P_5_B_2 TO P_5_TO_LOAD
  := FM_ZONE_4_SENSOR_2;
END_TRANSITION
END_ACTION
END_PROGRAM

CONFIGURATION Device
  RESOURCE Application ON PLC
    TASK MainTask(INTERVAL := T#20ms, PRIORITY := 1);
    PROGRAM PLC_PRG WITH MainTask : PLC_PRG;
  END_RESOURCE
END_CONFIGURATION
